// TIA Portal V20 export
// export: Created 2025-12-01T14:57:31.8385946Z, ExportSetting None, DisplayName Totally Integrated Automation Portal, DisplayVersion V20 Update 3, DisplayName TIA Portal Openness, DisplayVersion V20 Update 3, DisplayName TIA Portal Version Control Interface, DisplayVersion V20 Update 3, DisplayName STEP 7 Professional, DisplayVersion V20 Update 3, DisplayName STEP 7 Safety, DisplayVersion V20 Update 2, DisplayName WinCC Basic/Comfort/Advanced, DisplayVersion V20 Update 3, DisplayName WinCC Professional, DisplayVersion V20 Update 3, DisplayName WinCC Unified, DisplayVersion V20 Update 3
FUNCTION_BLOCK "FB531_Ordenes_ELEV / VTD"   // FB531, LAD
{ S7_Optimized_Access := 'FALSE' }
// stored: AutoNumber false, SetENOAutomatically false
   VAR_INPUT
      Estado_CBx : "EstadoZona";   // Estado de la Zona
      Maquina { ExternalVisible := 'False'; ExternalWritable := 'False'} : UInt;   // Numero de Máquina
      Error_Tx : Bool;
   END_VAR
   VAR_OUTPUT
      PosicionDestino : Real;
      Orden : Bool;
   END_VAR
   VAR
      PeticionPiso_Activa { ExternalAccessible := 'False'; ExternalVisible := 'False'; ExternalWritable := 'False'} : Bool;
      Mesa_AVTF_Activo : UInt;
      Mesa_DeDescarga : UInt;
      Mesa { ExternalAccessible := 'False'; ExternalVisible := 'False'; ExternalWritable := 'False'} : UInt;
      Mesa_H1 { ExternalAccessible := 'False'; ExternalVisible := 'False'; ExternalWritable := 'False'} : Bool;   // Orden de Descarga Horquilla/Mesa 1
      Mesa_H2 { ExternalAccessible := 'False'; ExternalVisible := 'False'; ExternalWritable := 'False'} : Bool;   // Orden de Descarga Horquilla/Mesa 2
      AVTF_Activo { ExternalAccessible := 'False'; ExternalVisible := 'False'; ExternalWritable := 'False'} : Bool;   // Orden de Carga hacia la Máquina
      OperacionJdT : Bool;
      Posicion_Destino { ExternalAccessible := 'False'; ExternalVisible := 'False'; ExternalWritable := 'False'} : Real;
      MesaDestino : UInt;
      Rem_MesaDestino : UInt;
      Rem_MesaOrigen : UInt;
   END_VAR
   VAR_TEMP
      OrdenJdT : Struct
         Operacion : UInt;
         MesaHorquilla : UInt;
         MesaCargaDesCarga : UInt;
         VarMesaHorquilla : UInt;
         VarMesaCargaDesCarga : UInt;
      END_STRUCT;
      PrimeraUT_EnMesa : UInt;
      NumMaquina : UInt;
      Mesa_1 : UInt;   // Horquilla/Mesa 1 de la máquina
      Mesa_2 : UInt;   // Horquilla/Mesa 2 de la máquina
      Cero : Byte;
      ValorReturn : Int;
   END_VAR
   VAR_TEMP   // added for the SCL form of the ladder/FBD networks
      _w1 : Bool;
      _w2 : Bool;
      _w3 : Bool;
   END_VAR
BEGIN

REGION Network 1 (SCL): INICIALIZACION
   #Posicion_Destino := 0;

   // Incializar temporales
   #PrimeraUT_EnMesa := 0;

   // Configugracion 
   #Mesa_1 := #NumMaquina :="DB885_ConfigMaquinas".Maquina[#Maquina].Mesa_1;
   #Mesa_2 := "DB885_ConfigMaquinas".Maquina[#Maquina].Mesa_2;

   /// Recoger ordens de JdT
   #OrdenJdT.Operacion := "DB832_Maquinas".Maquinas[#NumMaquina].VTD_ELEV.Operacion;
   #OrdenJdT.MesaHorquilla := "DB832_Maquinas".Maquinas[#NumMaquina].VTD_ELEV.MesaHorquilla ;
   #OrdenJdT.MesaCargaDesCarga := "DB832_Maquinas".Maquinas[#NumMaquina].VTD_ELEV.MesaCargaDesCarga;
   #OrdenJdT.VarMesaHorquilla := #OrdenJdT.MesaHorquilla - "CTE_OffsetMesa";
   #OrdenJdT.VarMesaCargaDesCarga := #OrdenJdT.MesaCargaDesCarga - "CTE_OffsetMesa";
END_REGION

REGION Network 2: >>>>>>>>>>>>>>>>>>>>>>>>>>>>>>>>>>>>>>>>>>>>>>>>>>>>>>>>>>>>>>>>>>>>>>>>>>>>>>>>
END_REGION

REGION Network 3 (SCL): CARGA DEL VTD
   //Si la zona no esta en Marcha o alguna mesa de la maquina esta en error -> No se hace nada 
   IF #Estado_CBx.Marcha_CBx AND #Error_Tx = FALSE THEN
       FOR #Mesa := 1 TO 500 BY 1 DO

           //Si se esta ejecutando una orden anterior no hacemos nada
           IF ((#OperacionJdT = FALSE) AND (#AVTF_Activo = FALSE) AND (#Mesa_H1 = FALSE) AND (#Mesa_H2 = FALSE)) THEN

               // Repasamos todas las mesas de acometida por si alguna tiene activo el AVTF     
               IF (("DB951_InterlockMaquinas".Maquina[#Maquina].Mesa[#Mesa].Out.AVTF) AND ("DB951_InterlockMaquinas".Maquina[#Maquina].Mesa[#Mesa].PosOK_H1 = FALSE) AND ("DB951_InterlockMaquinas".Maquina[#Maquina].Mesa[#Mesa].PosOK_H2 = FALSE)) THEN
                   #PrimeraUT_EnMesa := "DB810_ColasMesas".Colas[#Mesa_AVTF_Activo].UT_PrimeraMesa;
                   #MesaDestino := "DB812_UTs_Control".UT[#PrimeraUT_EnMesa].MesaDestino - "CTE_OffsetMesa";

                   // Revisamos si la mesa destino esta vacia
                   IF "DB900_Estado_Mesas".EstadoVI[#MesaDestino].Etapa_Vacia THEN
                       #Mesa_AVTF_Activo := #Mesa; // Guardamos la mesa que tiene el Aviso Activo
                       #AVTF_Activo := TRUE; 
                       EXIT;
                   END_IF;

               END_IF;
           END_IF;
       END_FOR;
   END_IF;
END_REGION

REGION Network 4: RESETEO SEÑALES CARGA DEL VTD
   // Si en una de las horquillas hay un error y la mesa de Destino se carga mientras resolvemos el error hay que resetear también.
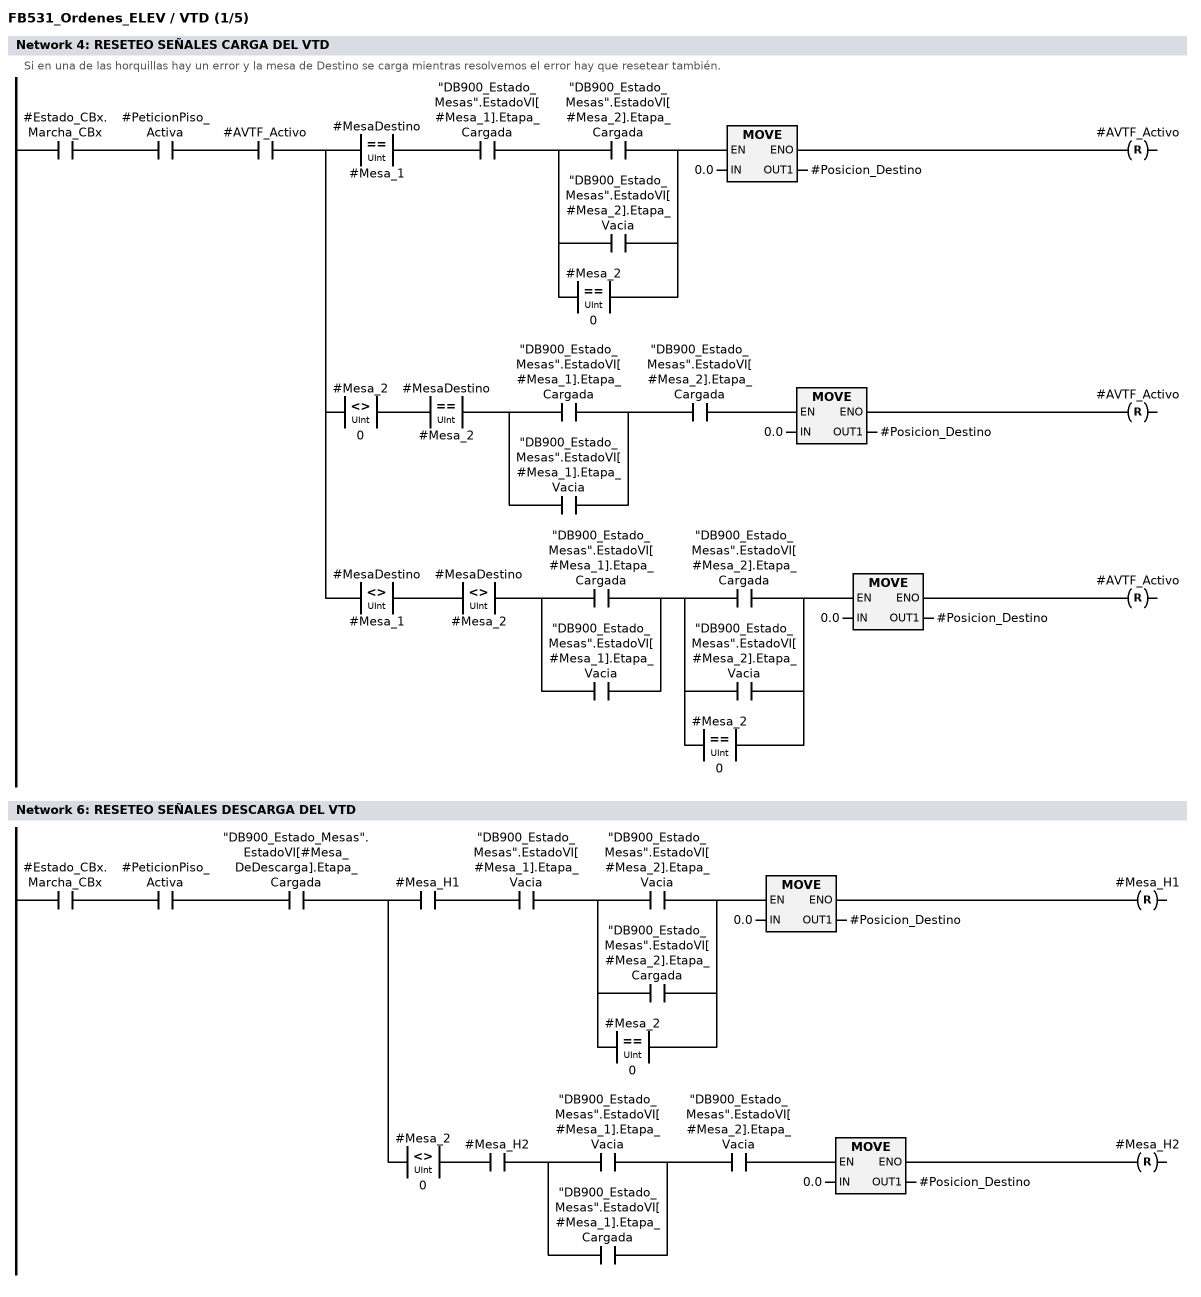
   RUNG wire#powerrail
      Contact( #Estado_CBx.Marcha_CBx )
      Contact( #PeticionPiso_Activa )
      Contact( #AVTF_Activo )
      wire#w1
      { S7_Templates := "SrcType := UInt" } EQ_Contact(in1 := #MesaDestino, in2 := #Mesa_1)
      Contact( "DB900_Estado_Mesas".EstadoVI[#Mesa_1].Etapa_Cargada )
      wire#w2
      Contact( "DB900_Estado_Mesas".EstadoVI[#Mesa_2].Etapa_Cargada )
      wire#w3
      Move(in := 0.0, out1 => #Posicion_Destino)
      R_Coil( #AVTF_Activo )
   END_RUNG
   RUNG wire#w2
      Contact( "DB900_Estado_Mesas".EstadoVI[#Mesa_2].Etapa_Vacia )
   END_RUNG wire#w3
   RUNG wire#w2
      { S7_Templates := "SrcType := UInt" } EQ_Contact(in1 := #Mesa_2, in2 := 0)
   END_RUNG wire#w3
   RUNG wire#w1
      { S7_Templates := "SrcType := UInt" } NE_Contact(in1 := #Mesa_2, in2 := 0)
      { S7_Templates := "SrcType := UInt" } EQ_Contact(in1 := #MesaDestino, in2 := #Mesa_2)
      wire#w4
      Contact( "DB900_Estado_Mesas".EstadoVI[#Mesa_1].Etapa_Cargada )
      wire#w5
      Contact( "DB900_Estado_Mesas".EstadoVI[#Mesa_2].Etapa_Cargada )
      Move(in := 0.0, out1 => #Posicion_Destino)
      R_Coil( #AVTF_Activo )
   END_RUNG
   RUNG wire#w4
      Contact( "DB900_Estado_Mesas".EstadoVI[#Mesa_1].Etapa_Vacia )
   END_RUNG wire#w5
   RUNG wire#w1
      { S7_Templates := "SrcType := UInt" } NE_Contact(in1 := #MesaDestino, in2 := #Mesa_1)
      { S7_Templates := "SrcType := UInt" } NE_Contact(in1 := #MesaDestino, in2 := #Mesa_2)
      wire#w6
      Contact( "DB900_Estado_Mesas".EstadoVI[#Mesa_1].Etapa_Cargada )
      wire#w7
      Contact( "DB900_Estado_Mesas".EstadoVI[#Mesa_2].Etapa_Cargada )
      wire#w8
      Move(in := 0.0, out1 => #Posicion_Destino)
      R_Coil( #AVTF_Activo )
   END_RUNG
   RUNG wire#w6
      Contact( "DB900_Estado_Mesas".EstadoVI[#Mesa_1].Etapa_Vacia )
   END_RUNG wire#w7
   RUNG wire#w7
      Contact( "DB900_Estado_Mesas".EstadoVI[#Mesa_2].Etapa_Vacia )
   END_RUNG wire#w8
   RUNG wire#w7
      { S7_Templates := "SrcType := UInt" } EQ_Contact(in1 := #Mesa_2, in2 := 0)
   END_RUNG wire#w8
   // the same network as SCL:
   #_w1 := #Estado_CBx.Marcha_CBx AND #PeticionPiso_Activa AND #AVTF_Activo;
   IF #_w1 AND (#MesaDestino = #Mesa_1) AND "DB900_Estado_Mesas".EstadoVI[#Mesa_1].Etapa_Cargada AND ("DB900_Estado_Mesas".EstadoVI[#Mesa_2].Etapa_Cargada OR "DB900_Estado_Mesas".EstadoVI[#Mesa_2].Etapa_Vacia OR (#Mesa_2 = 0)) THEN
       #Posicion_Destino := 0.0;
       #AVTF_Activo := FALSE;
   END_IF;
   IF #_w1 AND (#Mesa_2 <> 0) AND (#MesaDestino = #Mesa_2) AND ("DB900_Estado_Mesas".EstadoVI[#Mesa_1].Etapa_Cargada OR "DB900_Estado_Mesas".EstadoVI[#Mesa_1].Etapa_Vacia) AND "DB900_Estado_Mesas".EstadoVI[#Mesa_2].Etapa_Cargada THEN
       #Posicion_Destino := 0.0;
       #AVTF_Activo := FALSE;
   END_IF;
   IF #_w1 AND (#MesaDestino <> #Mesa_1) AND (#MesaDestino <> #Mesa_2) AND ("DB900_Estado_Mesas".EstadoVI[#Mesa_1].Etapa_Cargada OR "DB900_Estado_Mesas".EstadoVI[#Mesa_1].Etapa_Vacia) AND ("DB900_Estado_Mesas".EstadoVI[#Mesa_2].Etapa_Cargada OR "DB900_Estado_Mesas".EstadoVI[#Mesa_2].Etapa_Vacia OR (#Mesa_2 = 0)) THEN
       #Posicion_Destino := 0.0;
       #AVTF_Activo := FALSE;
   END_IF;
END_REGION

REGION Network 5 (SCL): DESCARGA DEL VTD
   //Si la zona no esta en Marcha o alguna mesa de la maquina esta en error -> No se hace nada 
   IF #Estado_CBx.Marcha_CBx = TRUE AND #Error_Tx = FALSE THEN

       //Si se esta ejecutando una orden anterior no hacemos nada
       IF ((#OperacionJdT = FALSE) AND (#AVTF_Activo = FALSE) AND (#Mesa_H1 = FALSE) AND (#Mesa_H2 = FALSE)) THEN

           // Repasamos todas las mesas de acometida por si alguna tiene activo el AVTF     
           IF (("DB900_Estado_Mesas".EstadoVI[#Mesa_1].Etapa_Cargada) AND ("DB951_InterlockMaquinas".Maquina[#Maquina].H1.Out.AVTF_Dcha OR "DB951_InterlockMaquinas".Maquina[#Maquina].H1.Out.AVTF_Izq)) THEN
               #PrimeraUT_EnMesa := "DB810_ColasMesas".Colas[#Mesa_1].UT_PrimeraMesa;
               #Mesa_DeDescarga := "DB812_UTs_Control".UT[#PrimeraUT_EnMesa].MesaDestino - "CTE_OffsetMesa";

               // Revisamos si la mesa destino esta vacia
               IF "DB900_Estado_Mesas".EstadoVI[#Mesa_DeDescarga].Etapa_Vacia THEN
                   #Mesa_H1 := TRUE;
               END_IF;

           ELSIF (("DB900_Estado_Mesas".EstadoVI[#Mesa_2].Etapa_Cargada) AND ("DB951_InterlockMaquinas".Maquina[#Maquina].H2.Out.AVTF_Dcha OR "DB951_InterlockMaquinas".Maquina[#Maquina].H2.Out.AVTF_Izq)) THEN
               #PrimeraUT_EnMesa := "DB810_ColasMesas".Colas[#Mesa_2].UT_PrimeraMesa;
               #Mesa_DeDescarga := "DB812_UTs_Control".UT[#PrimeraUT_EnMesa].MesaDestino - "CTE_OffsetMesa";

               // Revisamos si la mesa destino esta vacia
               IF "DB900_Estado_Mesas".EstadoVI[#Mesa_DeDescarga].Etapa_Vacia THEN
                   #Mesa_H2 := TRUE;
               END_IF;

           END_IF;
       END_IF;
   END_IF;
END_REGION

REGION Network 6: RESETEO SEÑALES DESCARGA DEL VTD
   RUNG wire#powerrail
      Contact( #Estado_CBx.Marcha_CBx )
      Contact( #PeticionPiso_Activa )
      Contact( "DB900_Estado_Mesas".EstadoVI[#Mesa_DeDescarga].Etapa_Cargada )
      wire#w1
      Contact( #Mesa_H1 )
      Contact( "DB900_Estado_Mesas".EstadoVI[#Mesa_1].Etapa_Vacia )
      wire#w2
      Contact( "DB900_Estado_Mesas".EstadoVI[#Mesa_2].Etapa_Vacia )
      wire#w3
      Move(in := 0.0, out1 => #Posicion_Destino)
      R_Coil( #Mesa_H1 )
   END_RUNG
   RUNG wire#w2
      Contact( "DB900_Estado_Mesas".EstadoVI[#Mesa_2].Etapa_Cargada )
   END_RUNG wire#w3
   RUNG wire#w2
      { S7_Templates := "SrcType := UInt" } EQ_Contact(in1 := #Mesa_2, in2 := 0)
   END_RUNG wire#w3
   RUNG wire#w1
      { S7_Templates := "SrcType := UInt" } NE_Contact(in1 := #Mesa_2, in2 := 0)
      Contact( #Mesa_H2 )
      wire#w4
      Contact( "DB900_Estado_Mesas".EstadoVI[#Mesa_1].Etapa_Vacia )
      wire#w5
      Contact( "DB900_Estado_Mesas".EstadoVI[#Mesa_2].Etapa_Vacia )
      Move(in := 0.0, out1 => #Posicion_Destino)
      R_Coil( #Mesa_H2 )
   END_RUNG
   RUNG wire#w4
      Contact( "DB900_Estado_Mesas".EstadoVI[#Mesa_1].Etapa_Cargada )
   END_RUNG wire#w5
   // the same network as SCL:
   #_w1 := #Estado_CBx.Marcha_CBx AND #PeticionPiso_Activa AND "DB900_Estado_Mesas".EstadoVI[#Mesa_DeDescarga].Etapa_Cargada;
   IF #_w1 AND #Mesa_H1 AND "DB900_Estado_Mesas".EstadoVI[#Mesa_1].Etapa_Vacia AND ("DB900_Estado_Mesas".EstadoVI[#Mesa_2].Etapa_Vacia OR "DB900_Estado_Mesas".EstadoVI[#Mesa_2].Etapa_Cargada OR (#Mesa_2 = 0)) THEN
       #Posicion_Destino := 0.0;
       #Mesa_H1 := FALSE;
   END_IF;
   IF #_w1 AND (#Mesa_2 <> 0) AND #Mesa_H2 AND ("DB900_Estado_Mesas".EstadoVI[#Mesa_1].Etapa_Vacia OR "DB900_Estado_Mesas".EstadoVI[#Mesa_1].Etapa_Cargada) AND "DB900_Estado_Mesas".EstadoVI[#Mesa_2].Etapa_Vacia THEN
       #Posicion_Destino := 0.0;
       #Mesa_H2 := FALSE;
   END_IF;
END_REGION

REGION Network 7: >>>>>>>>>>>>>>>>>>>>>>>>>>>>>>>>>>>>>>>>>>>>>>>>>>>>>>>>>>>>>>>>>>>>>>>>>>>>>>>>
END_REGION

REGION Network 8: Activamos las peticiones para mover la maquina
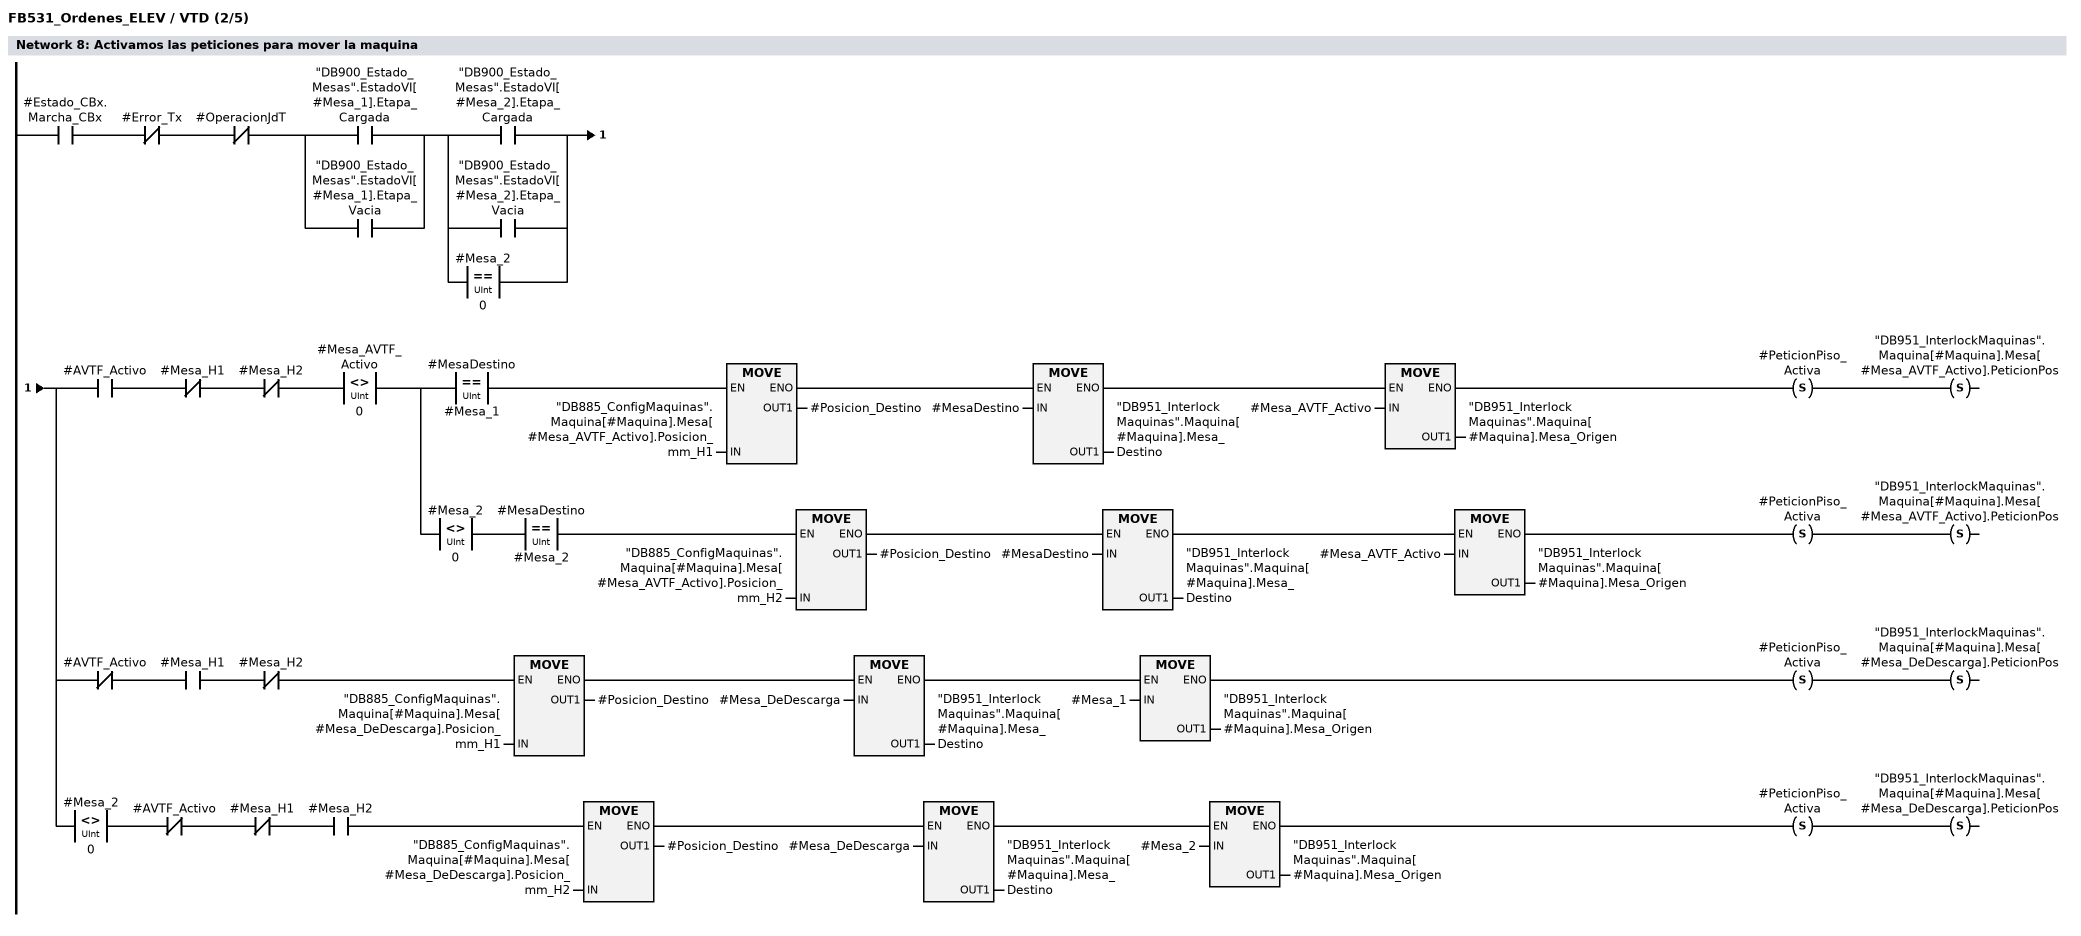
   RUNG wire#powerrail
      Contact( #Estado_CBx.Marcha_CBx )
      I_Contact( #Error_Tx )
      I_Contact( #OperacionJdT )
      wire#w1
      Contact( "DB900_Estado_Mesas".EstadoVI[#Mesa_1].Etapa_Cargada )
      wire#w2
      Contact( "DB900_Estado_Mesas".EstadoVI[#Mesa_2].Etapa_Cargada )
      wire#w3
      Contact( #AVTF_Activo )
      I_Contact( #Mesa_H1 )
      I_Contact( #Mesa_H2 )
      { S7_Templates := "SrcType := UInt" } NE_Contact(in1 := #Mesa_AVTF_Activo, in2 := 0)
      wire#w4
      { S7_Templates := "SrcType := UInt" } EQ_Contact(in1 := #MesaDestino, in2 := #Mesa_1)
      Move(in := "DB885_ConfigMaquinas".Maquina[#Maquina].Mesa[#Mesa_AVTF_Activo].Posicion_mm_H1, out1 => #Posicion_Destino)
      Move(in := #MesaDestino, out1 => "DB951_InterlockMaquinas".Maquina[#Maquina].Mesa_Destino)
      Move(in := #Mesa_AVTF_Activo, out1 => "DB951_InterlockMaquinas".Maquina[#Maquina].Mesa_Origen)
      S_Coil( #PeticionPiso_Activa )
      S_Coil( "DB951_InterlockMaquinas".Maquina[#Maquina].Mesa[#Mesa_AVTF_Activo].PeticionPos )
   END_RUNG
   RUNG wire#w1
      Contact( "DB900_Estado_Mesas".EstadoVI[#Mesa_1].Etapa_Vacia )
   END_RUNG wire#w2
   RUNG wire#w2
      Contact( "DB900_Estado_Mesas".EstadoVI[#Mesa_2].Etapa_Vacia )
   END_RUNG wire#w3
   RUNG wire#w2
      { S7_Templates := "SrcType := UInt" } EQ_Contact(in1 := #Mesa_2, in2 := 0)
   END_RUNG wire#w3
   RUNG wire#w4
      { S7_Templates := "SrcType := UInt" } NE_Contact(in1 := #Mesa_2, in2 := 0)
      { S7_Templates := "SrcType := UInt" } EQ_Contact(in1 := #MesaDestino, in2 := #Mesa_2)
      Move(in := "DB885_ConfigMaquinas".Maquina[#Maquina].Mesa[#Mesa_AVTF_Activo].Posicion_mm_H2, out1 => #Posicion_Destino)
      Move(in := #MesaDestino, out1 => "DB951_InterlockMaquinas".Maquina[#Maquina].Mesa_Destino)
      Move(in := #Mesa_AVTF_Activo, out1 => "DB951_InterlockMaquinas".Maquina[#Maquina].Mesa_Origen)
      S_Coil( #PeticionPiso_Activa )
      S_Coil( "DB951_InterlockMaquinas".Maquina[#Maquina].Mesa[#Mesa_AVTF_Activo].PeticionPos )
   END_RUNG
   RUNG wire#w3
      I_Contact( #AVTF_Activo )
      Contact( #Mesa_H1 )
      I_Contact( #Mesa_H2 )
      Move(in := "DB885_ConfigMaquinas".Maquina[#Maquina].Mesa[#Mesa_DeDescarga].Posicion_mm_H1, out1 => #Posicion_Destino)
      Move(in := #Mesa_DeDescarga, out1 => "DB951_InterlockMaquinas".Maquina[#Maquina].Mesa_Destino)
      Move(in := #Mesa_1, out1 => "DB951_InterlockMaquinas".Maquina[#Maquina].Mesa_Origen)
      S_Coil( #PeticionPiso_Activa )
      S_Coil( "DB951_InterlockMaquinas".Maquina[#Maquina].Mesa[#Mesa_DeDescarga].PeticionPos )
   END_RUNG
   RUNG wire#w3
      { S7_Templates := "SrcType := UInt" } NE_Contact(in1 := #Mesa_2, in2 := 0)
      I_Contact( #AVTF_Activo )
      I_Contact( #Mesa_H1 )
      Contact( #Mesa_H2 )
      Move(in := "DB885_ConfigMaquinas".Maquina[#Maquina].Mesa[#Mesa_DeDescarga].Posicion_mm_H2, out1 => #Posicion_Destino)
      Move(in := #Mesa_DeDescarga, out1 => "DB951_InterlockMaquinas".Maquina[#Maquina].Mesa_Destino)
      Move(in := #Mesa_2, out1 => "DB951_InterlockMaquinas".Maquina[#Maquina].Mesa_Origen)
      S_Coil( #PeticionPiso_Activa )
      S_Coil( "DB951_InterlockMaquinas".Maquina[#Maquina].Mesa[#Mesa_DeDescarga].PeticionPos )
   END_RUNG
   // the same network as SCL:
   #_w1 := #Estado_CBx.Marcha_CBx AND NOT #Error_Tx AND NOT #OperacionJdT AND ("DB900_Estado_Mesas".EstadoVI[#Mesa_1].Etapa_Cargada OR "DB900_Estado_Mesas".EstadoVI[#Mesa_1].Etapa_Vacia) AND ("DB900_Estado_Mesas".EstadoVI[#Mesa_2].Etapa_Cargada OR "DB900_Estado_Mesas".EstadoVI[#Mesa_2].Etapa_Vacia OR (#Mesa_2 = 0));
   #_w2 := #_w1 AND #AVTF_Activo AND NOT #Mesa_H1 AND NOT #Mesa_H2 AND (#Mesa_AVTF_Activo <> 0);
   IF #_w2 AND (#MesaDestino = #Mesa_1) THEN
       #Posicion_Destino := "DB885_ConfigMaquinas".Maquina[#Maquina].Mesa[#Mesa_AVTF_Activo].Posicion_mm_H1;
       "DB951_InterlockMaquinas".Maquina[#Maquina].Mesa_Destino := #MesaDestino;
       "DB951_InterlockMaquinas".Maquina[#Maquina].Mesa_Origen := #Mesa_AVTF_Activo;
       #PeticionPiso_Activa := TRUE;
       "DB951_InterlockMaquinas".Maquina[#Maquina].Mesa[#Mesa_AVTF_Activo].PeticionPos := TRUE;
   END_IF;
   IF #_w2 AND (#Mesa_2 <> 0) AND (#MesaDestino = #Mesa_2) THEN
       #Posicion_Destino := "DB885_ConfigMaquinas".Maquina[#Maquina].Mesa[#Mesa_AVTF_Activo].Posicion_mm_H2;
       "DB951_InterlockMaquinas".Maquina[#Maquina].Mesa_Destino := #MesaDestino;
       "DB951_InterlockMaquinas".Maquina[#Maquina].Mesa_Origen := #Mesa_AVTF_Activo;
       #PeticionPiso_Activa := TRUE;
       "DB951_InterlockMaquinas".Maquina[#Maquina].Mesa[#Mesa_AVTF_Activo].PeticionPos := TRUE;
   END_IF;
   IF #_w1 AND NOT #AVTF_Activo AND #Mesa_H1 AND NOT #Mesa_H2 THEN
       #Posicion_Destino := "DB885_ConfigMaquinas".Maquina[#Maquina].Mesa[#Mesa_DeDescarga].Posicion_mm_H1;
       "DB951_InterlockMaquinas".Maquina[#Maquina].Mesa_Destino := #Mesa_DeDescarga;
       "DB951_InterlockMaquinas".Maquina[#Maquina].Mesa_Origen := #Mesa_1;
       #PeticionPiso_Activa := TRUE;
       "DB951_InterlockMaquinas".Maquina[#Maquina].Mesa[#Mesa_DeDescarga].PeticionPos := TRUE;
   END_IF;
   IF #_w1 AND (#Mesa_2 <> 0) AND NOT #AVTF_Activo AND NOT #Mesa_H1 AND #Mesa_H2 THEN
       #Posicion_Destino := "DB885_ConfigMaquinas".Maquina[#Maquina].Mesa[#Mesa_DeDescarga].Posicion_mm_H2;
       "DB951_InterlockMaquinas".Maquina[#Maquina].Mesa_Destino := #Mesa_DeDescarga;
       "DB951_InterlockMaquinas".Maquina[#Maquina].Mesa_Origen := #Mesa_2;
       #PeticionPiso_Activa := TRUE;
       "DB951_InterlockMaquinas".Maquina[#Maquina].Mesa[#Mesa_DeDescarga].PeticionPos := TRUE;
   END_IF;
END_REGION

REGION Network 9: >>>>>>>>>>>>>>>>>>>>>>>>>>>>>>>>>>>>>>>>>>>>>>>>>>>>>>>>>>>>>>>>>>>>>>>>>>>>>>>>
END_REGION

REGION Network 10: SET >>> Operaciones desde JDT
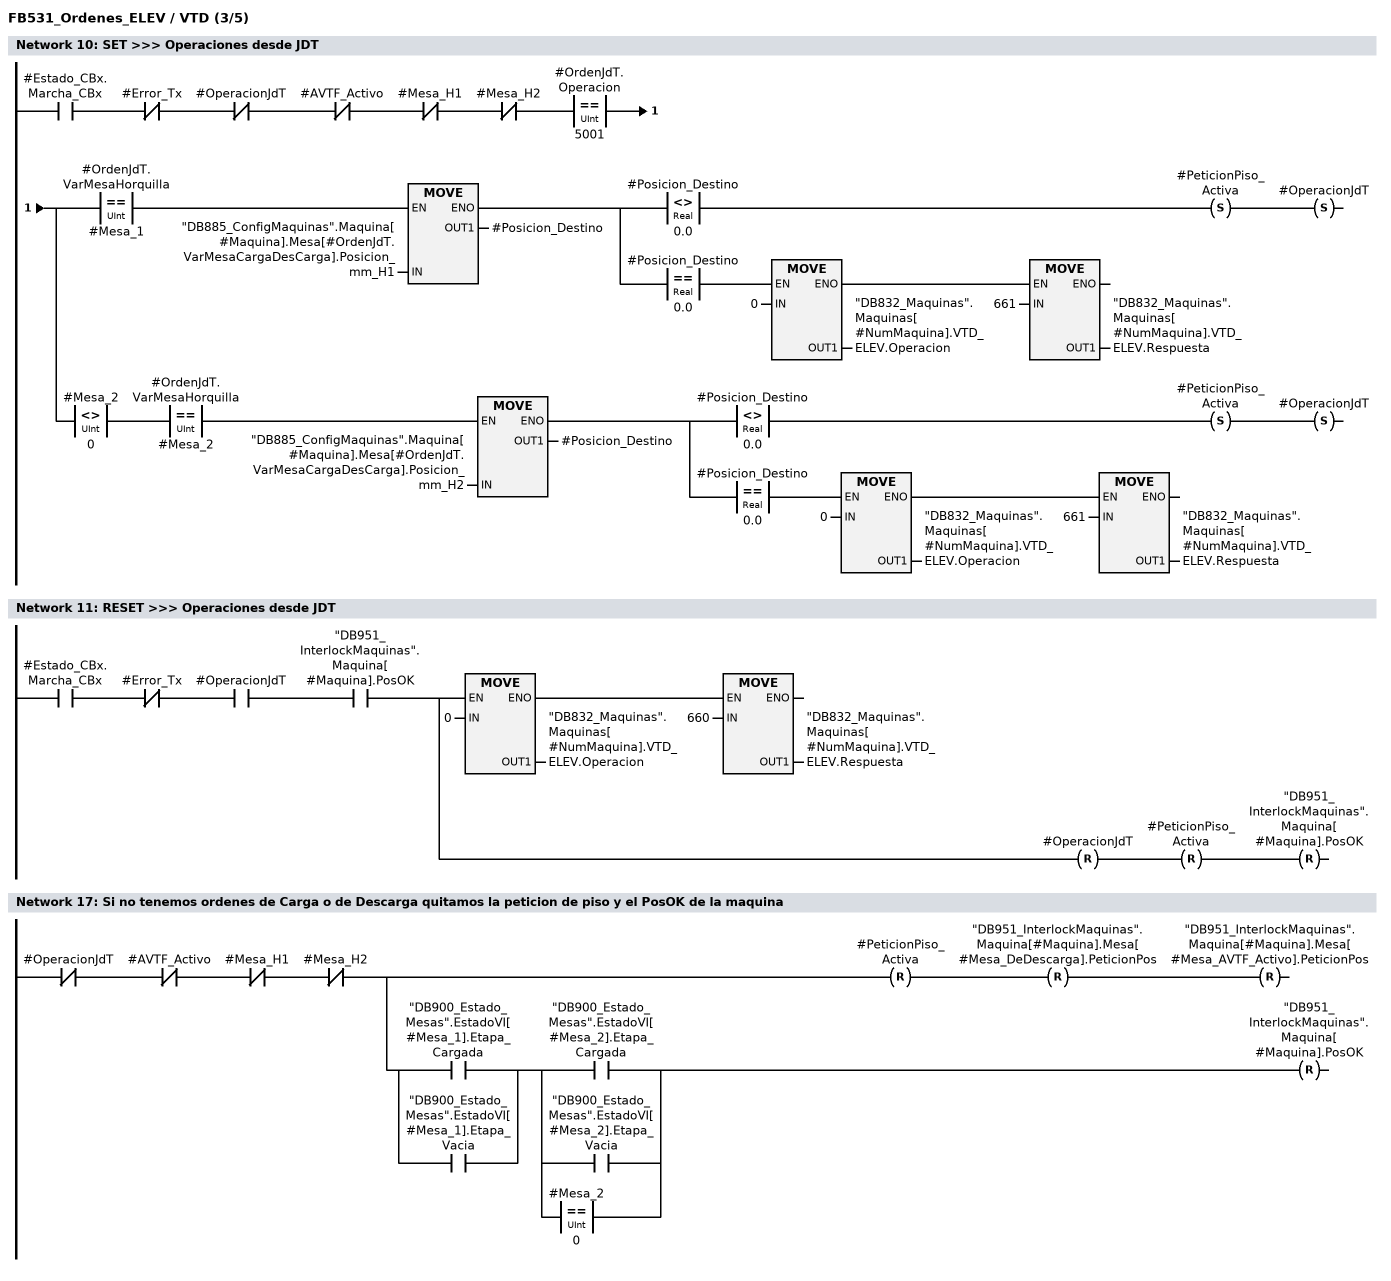
   RUNG wire#powerrail
      Contact( #Estado_CBx.Marcha_CBx )
      I_Contact( #Error_Tx )
      I_Contact( #OperacionJdT )
      I_Contact( #AVTF_Activo )
      I_Contact( #Mesa_H1 )
      I_Contact( #Mesa_H2 )
      { S7_Templates := "SrcType := UInt" } EQ_Contact(in1 := #OrdenJdT.Operacion, in2 := 5001)
      wire#w1
      { S7_Templates := "SrcType := UInt" } EQ_Contact(in1 := #OrdenJdT.VarMesaHorquilla, in2 := #Mesa_1)
      Move(in := "DB885_ConfigMaquinas".Maquina[#Maquina].Mesa[#OrdenJdT.VarMesaCargaDesCarga].Posicion_mm_H1, out1 => #Posicion_Destino)
      wire#w2
      { S7_Templates := "SrcType := Real" } NE_Contact(in1 := #Posicion_Destino, in2 := 0.0)
      S_Coil( #PeticionPiso_Activa )
      S_Coil( #OperacionJdT )
   END_RUNG
   RUNG wire#w2
      { S7_Templates := "SrcType := Real" } EQ_Contact(in1 := #Posicion_Destino, in2 := 0.0)
      Move(in := 0, out1 => "DB832_Maquinas".Maquinas[#NumMaquina].VTD_ELEV.Operacion)
      Move(in := 661, out1 => "DB832_Maquinas".Maquinas[#NumMaquina].VTD_ELEV.Respuesta)
   END_RUNG
   RUNG wire#w1
      { S7_Templates := "SrcType := UInt" } NE_Contact(in1 := #Mesa_2, in2 := 0)
      { S7_Templates := "SrcType := UInt" } EQ_Contact(in1 := #OrdenJdT.VarMesaHorquilla, in2 := #Mesa_2)
      Move(in := "DB885_ConfigMaquinas".Maquina[#Maquina].Mesa[#OrdenJdT.VarMesaCargaDesCarga].Posicion_mm_H2, out1 => #Posicion_Destino)
      wire#w3
      { S7_Templates := "SrcType := Real" } NE_Contact(in1 := #Posicion_Destino, in2 := 0.0)
      S_Coil( #PeticionPiso_Activa )
      S_Coil( #OperacionJdT )
   END_RUNG
   RUNG wire#w3
      { S7_Templates := "SrcType := Real" } EQ_Contact(in1 := #Posicion_Destino, in2 := 0.0)
      Move(in := 0, out1 => "DB832_Maquinas".Maquinas[#NumMaquina].VTD_ELEV.Operacion)
      Move(in := 661, out1 => "DB832_Maquinas".Maquinas[#NumMaquina].VTD_ELEV.Respuesta)
   END_RUNG
   // the same network as SCL:
   #_w1 := #Estado_CBx.Marcha_CBx AND NOT #Error_Tx AND NOT #OperacionJdT AND NOT #AVTF_Activo AND NOT #Mesa_H1 AND NOT #Mesa_H2 AND (#OrdenJdT.Operacion = 5001);
   #_w2 := #_w1 AND (#OrdenJdT.VarMesaHorquilla = #Mesa_1);
   IF #_w2 THEN
       #Posicion_Destino := "DB885_ConfigMaquinas".Maquina[#Maquina].Mesa[#OrdenJdT.VarMesaCargaDesCarga].Posicion_mm_H1;
   END_IF;
   IF #_w2 AND (#Posicion_Destino <> 0.0) THEN
       #PeticionPiso_Activa := TRUE;
       #OperacionJdT := TRUE;
   END_IF;
   IF #_w2 AND (#Posicion_Destino = 0.0) THEN
       "DB832_Maquinas".Maquinas[#NumMaquina].VTD_ELEV.Operacion := 0;
       "DB832_Maquinas".Maquinas[#NumMaquina].VTD_ELEV.Respuesta := 661;
   END_IF;
   #_w3 := #_w1 AND (#Mesa_2 <> 0) AND (#OrdenJdT.VarMesaHorquilla = #Mesa_2);
   IF #_w3 THEN
       #Posicion_Destino := "DB885_ConfigMaquinas".Maquina[#Maquina].Mesa[#OrdenJdT.VarMesaCargaDesCarga].Posicion_mm_H2;
   END_IF;
   IF #_w3 AND (#Posicion_Destino <> 0.0) THEN
       #PeticionPiso_Activa := TRUE;
       #OperacionJdT := TRUE;
   END_IF;
   IF #_w3 AND (#Posicion_Destino = 0.0) THEN
       "DB832_Maquinas".Maquinas[#NumMaquina].VTD_ELEV.Operacion := 0;
       "DB832_Maquinas".Maquinas[#NumMaquina].VTD_ELEV.Respuesta := 661;
   END_IF;
END_REGION

REGION Network 11: RESET >>> Operaciones desde JDT
   RUNG wire#powerrail
      Contact( #Estado_CBx.Marcha_CBx )
      I_Contact( #Error_Tx )
      Contact( #OperacionJdT )
      Contact( "DB951_InterlockMaquinas".Maquina[#Maquina].PosOK )
      wire#w1
      Move(in := 0, out1 => "DB832_Maquinas".Maquinas[#NumMaquina].VTD_ELEV.Operacion)
      Move(in := 660, out1 => "DB832_Maquinas".Maquinas[#NumMaquina].VTD_ELEV.Respuesta)
   END_RUNG
   RUNG wire#w1
      R_Coil( #OperacionJdT )
      R_Coil( #PeticionPiso_Activa )
      R_Coil( "DB951_InterlockMaquinas".Maquina[#Maquina].PosOK )
   END_RUNG
   // the same network as SCL:
   IF #Estado_CBx.Marcha_CBx AND NOT #Error_Tx AND #OperacionJdT AND "DB951_InterlockMaquinas".Maquina[#Maquina].PosOK THEN
       "DB832_Maquinas".Maquinas[#NumMaquina].VTD_ELEV.Operacion := 0;
       "DB832_Maquinas".Maquinas[#NumMaquina].VTD_ELEV.Respuesta := 660;
   END_IF;
   #_w1 := #Estado_CBx.Marcha_CBx AND NOT #Error_Tx AND #OperacionJdT AND "DB951_InterlockMaquinas".Maquina[#Maquina].PosOK;
   IF #_w1 THEN
       #OperacionJdT := FALSE;
       #PeticionPiso_Activa := FALSE;
       "DB951_InterlockMaquinas".Maquina[#Maquina].PosOK := FALSE;
   END_IF;
END_REGION

REGION Network 12: >>>>>>>>>>>>>>>>>>>>>>>>>>>>>>>>>>>>>>>>>>>>>>>>>>>>>>>>>>>>>>>>>>>>>>>>>>>>>>>>
END_REGION

REGION Network 13 (SCL): Inicializar interlock de la maquina

   #Cero := 0;

   #ValorReturn := FILL(BVAL := #Cero, BLK => "DB951_InterlockMaquinas".Maquina[#Maquina].H1.In);
   #ValorReturn := FILL(BVAL := #Cero, BLK => "DB951_InterlockMaquinas".Maquina[#Maquina].H2.In);

   "DB951_InterlockMaquinas".Maquina[#Maquina].H1.Mesa_EntradaDerecha := 0;
   "DB951_InterlockMaquinas".Maquina[#Maquina].H1.Mesa_EntradaIzquierda := 0;
   "DB951_InterlockMaquinas".Maquina[#Maquina].H2.Mesa_EntradaDerecha := 0;
   "DB951_InterlockMaquinas".Maquina[#Maquina].H2.Mesa_EntradaIzquierda := 0;
END_REGION

REGION Network 14 (SCL): Señales para cargar las mesas de la maquina
   FOR #Mesa := 1 TO 500 BY 1 DO

       #ValorReturn := FILL(BVAL := #Cero, BLK => "DB951_InterlockMaquinas".Maquina[#Maquina].Mesa[#Mesa].In);

         IF "DB951_InterlockMaquinas".Maquina[#Maquina].PosOK THEN
               // Repasamos que mesas tienen la misma cota para la Horquilla 1
               IF "DB885_ConfigMaquinas".Maquina[#Maquina].Mesa[#Mesa].Posicion_mm_H1 = #Posicion_Destino AND "DB951_InterlockMaquinas".Maquina[#Maquina].Mesa[#Mesa].PosOK_H1 THEN

                   // Señales de las Mesas posicionadas a la Derecha
                   IF "DB885_ConfigMaquinas".Maquina[#Maquina].Mesa[#Mesa].Derecha THEN
                       // Señales para cargar las mesas de la maquina
                       "DB951_InterlockMaquinas".Maquina[#Maquina].H1.In.AVTF_Dcha := "DB951_InterlockMaquinas".Maquina[#Maquina].Mesa[#Mesa].Out.AVTF;
                       "DB951_InterlockMaquinas".Maquina[#Maquina].H1.In.P_Mens_Dcha := "DB951_InterlockMaquinas".Maquina[#Maquina].Mesa[#Mesa].Out.P_Mens;
                       "DB951_InterlockMaquinas".Maquina[#Maquina].H1.In.DesCargaAct_Dcha := "DB900_Estado_Mesas".EstadoVI[#Mesa].Descarga_Act;

                       "DB951_InterlockMaquinas".Maquina[#Maquina].Mesa[#Mesa].In.PTF := "DB951_InterlockMaquinas".Maquina[#Maquina].H1.Out.PTF_Dcha;
                       "DB951_InterlockMaquinas".Maquina[#Maquina].Mesa[#Mesa].In.FTF := "DB951_InterlockMaquinas".Maquina[#Maquina].H1.Out.FTF_Dcha;
                       "DB951_InterlockMaquinas".Maquina[#Maquina].Mesa[#Mesa].In.CargaAct := "DB900_Estado_Mesas".EstadoVI[#Mesa_1].Etapas_Carga_E1;

                       "DB951_InterlockMaquinas".Maquina[#Maquina].H1.Mesa_EntradaDerecha := #Mesa;

                       // Señales para descargar las mesas de la maquina
                       "DB951_InterlockMaquinas".Maquina[#Maquina].Mesa[#Mesa].In.AVTF := "DB951_InterlockMaquinas".Maquina[#Maquina].H1.Out.AVTF_Dcha;
                       "DB951_InterlockMaquinas".Maquina[#Maquina].Mesa[#Mesa].In.P_Mens := "DB951_InterlockMaquinas".Maquina[#Maquina].H1.Out.P_Mens_Dcha;
                       "DB951_InterlockMaquinas".Maquina[#Maquina].Mesa[#Mesa].In.DesCargaAct := "DB900_Estado_Mesas".EstadoVI[#Mesa_1].Descarga_Act;

                       "DB951_InterlockMaquinas".Maquina[#Maquina].H1.In.PTF_Dcha := "DB951_InterlockMaquinas".Maquina[#Maquina].Mesa[#Mesa].Out.PTF;
                       "DB951_InterlockMaquinas".Maquina[#Maquina].H1.In.FTF_Dcha := "DB951_InterlockMaquinas".Maquina[#Maquina].Mesa[#Mesa].Out.FTF;
                       "DB951_InterlockMaquinas".Maquina[#Maquina].H1.In.CargaAct_Dcha := "DB900_Estado_Mesas".EstadoVI[#Mesa].Etapas_Carga_E1 OR
                                                                                               "DB900_Estado_Mesas".EstadoVI[#Mesa].Etapas_Carga_E2 OR
                                                                                               "DB900_Estado_Mesas".EstadoVI[#Mesa].Etapas_Carga_E3 OR
                                                                                               "DB900_Estado_Mesas".EstadoVI[#Mesa].Etapas_Carga_E4;

                       "DB951_InterlockMaquinas".Maquina[#Maquina].Mesa[#Mesa].MesaEntrada := #Mesa_1;

                   END_IF;

                   // Señales de las Mesas posicionadas a la Izquierda
                   IF "DB885_ConfigMaquinas".Maquina[#Maquina].Mesa[#Mesa].Izquierda THEN
                       // Señales para cargar las mesas de la maquina
                       "DB951_InterlockMaquinas".Maquina[#Maquina].H1.In.AVTF_Izq := "DB951_InterlockMaquinas".Maquina[#Maquina].Mesa[#Mesa].Out.AVTF;
                       "DB951_InterlockMaquinas".Maquina[#Maquina].H1.In.P_Mens_Izq := "DB951_InterlockMaquinas".Maquina[#Maquina].Mesa[#Mesa].Out.P_Mens;
                       "DB951_InterlockMaquinas".Maquina[#Maquina].H1.In.DesCargaAct_Izq := "DB900_Estado_Mesas".EstadoVI[#Mesa].Descarga_Act;

                       "DB951_InterlockMaquinas".Maquina[#Maquina].Mesa[#Mesa].In.PTF := "DB951_InterlockMaquinas".Maquina[#Maquina].H1.Out.PTF_Izq;
                       "DB951_InterlockMaquinas".Maquina[#Maquina].Mesa[#Mesa].In.FTF := "DB951_InterlockMaquinas".Maquina[#Maquina].H1.Out.FTF_Izq;
                       "DB951_InterlockMaquinas".Maquina[#Maquina].Mesa[#Mesa].In.CargaAct := "DB900_Estado_Mesas".EstadoVI[#Mesa_1].Etapas_Carga_E3;

                       "DB951_InterlockMaquinas".Maquina[#Maquina].H1.Mesa_EntradaIzquierda := #Mesa;

                       // Señales para descargar las mesas de la maquina
                       "DB951_InterlockMaquinas".Maquina[#Maquina].Mesa[#Mesa].In.AVTF := "DB951_InterlockMaquinas".Maquina[#Maquina].H1.Out.AVTF_Izq;
                       "DB951_InterlockMaquinas".Maquina[#Maquina].Mesa[#Mesa].In.P_Mens := "DB951_InterlockMaquinas".Maquina[#Maquina].H1.Out.P_Mens_Izq;
                       "DB951_InterlockMaquinas".Maquina[#Maquina].Mesa[#Mesa].In.DesCargaAct := "DB900_Estado_Mesas".EstadoVI[#Mesa_1].Descarga_Act;

                       "DB951_InterlockMaquinas".Maquina[#Maquina].H1.In.PTF_Izq := "DB951_InterlockMaquinas".Maquina[#Maquina].Mesa[#Mesa].Out.PTF;
                       "DB951_InterlockMaquinas".Maquina[#Maquina].H1.In.FTF_Izq := "DB951_InterlockMaquinas".Maquina[#Maquina].Mesa[#Mesa].Out.FTF;
                       "DB951_InterlockMaquinas".Maquina[#Maquina].H1.In.CargaAct_Izq := "DB900_Estado_Mesas".EstadoVI[#Mesa].Etapas_Carga_E1 OR
                                                                                               "DB900_Estado_Mesas".EstadoVI[#Mesa].Etapas_Carga_E2 OR
                                                                                               "DB900_Estado_Mesas".EstadoVI[#Mesa].Etapas_Carga_E3 OR
                                                                                               "DB900_Estado_Mesas".EstadoVI[#Mesa].Etapas_Carga_E4;

                       "DB951_InterlockMaquinas".Maquina[#Maquina].Mesa[#Mesa].MesaEntrada := #Mesa_1;
                   END_IF;

               END_IF;

               // Repasamos que mesas tienen la misma cota para la Horquilla 2
               IF "DB885_ConfigMaquinas".Maquina[#Maquina].Mesa[#Mesa].Posicion_mm_H2 = #Posicion_Destino AND "DB951_InterlockMaquinas".Maquina[#Maquina].Mesa[#Mesa].PosOK_H2 THEN

                   // Señales de las Mesas posicionadas a la Derecha
                   IF "DB885_ConfigMaquinas".Maquina[#Maquina].Mesa[#Mesa].Derecha THEN
                       // Señales para cargar las mesas de la maquina
                       "DB951_InterlockMaquinas".Maquina[#Maquina].H2.In.AVTF_Dcha := "DB951_InterlockMaquinas".Maquina[#Maquina].Mesa[#Mesa].Out.AVTF;
                       "DB951_InterlockMaquinas".Maquina[#Maquina].H2.In.P_Mens_Dcha := "DB951_InterlockMaquinas".Maquina[#Maquina].Mesa[#Mesa].Out.P_Mens;
                       "DB951_InterlockMaquinas".Maquina[#Maquina].H2.In.DesCargaAct_Dcha := "DB900_Estado_Mesas".EstadoVI[#Mesa].Descarga_Act;

                       "DB951_InterlockMaquinas".Maquina[#Maquina].Mesa[#Mesa].In.PTF := "DB951_InterlockMaquinas".Maquina[#Maquina].H2.Out.PTF_Dcha;
                       "DB951_InterlockMaquinas".Maquina[#Maquina].Mesa[#Mesa].In.FTF := "DB951_InterlockMaquinas".Maquina[#Maquina].H2.Out.FTF_Dcha;
                       "DB951_InterlockMaquinas".Maquina[#Maquina].Mesa[#Mesa].In.CargaAct := "DB900_Estado_Mesas".EstadoVI[#Mesa_2].Etapas_Carga_E1;

                       "DB951_InterlockMaquinas".Maquina[#Maquina].H2.Mesa_EntradaDerecha := #Mesa;

                       // Señales para descargar las mesas de la maquina
                       "DB951_InterlockMaquinas".Maquina[#Maquina].Mesa[#Mesa].In.AVTF := "DB951_InterlockMaquinas".Maquina[#Maquina].H2.Out.AVTF_Dcha;
                       "DB951_InterlockMaquinas".Maquina[#Maquina].Mesa[#Mesa].In.P_Mens := "DB951_InterlockMaquinas".Maquina[#Maquina].H2.Out.P_Mens_Dcha;
                       "DB951_InterlockMaquinas".Maquina[#Maquina].Mesa[#Mesa].In.DesCargaAct := "DB900_Estado_Mesas".EstadoVI[#Mesa_2].Descarga_Act;

                       "DB951_InterlockMaquinas".Maquina[#Maquina].H2.In.PTF_Dcha := "DB951_InterlockMaquinas".Maquina[#Maquina].Mesa[#Mesa].Out.PTF;
                       "DB951_InterlockMaquinas".Maquina[#Maquina].H2.In.FTF_Dcha := "DB951_InterlockMaquinas".Maquina[#Maquina].Mesa[#Mesa].Out.FTF;
                       "DB951_InterlockMaquinas".Maquina[#Maquina].H2.In.CargaAct_Dcha := "DB900_Estado_Mesas".EstadoVI[#Mesa].Etapas_Carga_E1 OR
                                                                                               "DB900_Estado_Mesas".EstadoVI[#Mesa].Etapas_Carga_E2 OR
                                                                                               "DB900_Estado_Mesas".EstadoVI[#Mesa].Etapas_Carga_E3 OR
                                                                                               "DB900_Estado_Mesas".EstadoVI[#Mesa].Etapas_Carga_E4;


                       "DB951_InterlockMaquinas".Maquina[#Maquina].Mesa[#Mesa].MesaEntrada := #Mesa_2;

                   END_IF;

                   // Señales de las Mesas posicionadas a la Izquierda
                   IF "DB885_ConfigMaquinas".Maquina[#Maquina].Mesa[#Mesa].Izquierda THEN
                       // Señales para cargar las mesas de la maquina
                       "DB951_InterlockMaquinas".Maquina[#Maquina].H2.In.AVTF_Izq := "DB951_InterlockMaquinas".Maquina[#Maquina].Mesa[#Mesa].Out.AVTF;
                       "DB951_InterlockMaquinas".Maquina[#Maquina].H2.In.P_Mens_Izq := "DB951_InterlockMaquinas".Maquina[#Maquina].Mesa[#Mesa].Out.P_Mens;
                       "DB951_InterlockMaquinas".Maquina[#Maquina].H2.In.DesCargaAct_Izq := "DB900_Estado_Mesas".EstadoVI[#Mesa].Descarga_Act;

                       "DB951_InterlockMaquinas".Maquina[#Maquina].Mesa[#Mesa].In.PTF := "DB951_InterlockMaquinas".Maquina[#Maquina].H2.Out.PTF_Izq;
                       "DB951_InterlockMaquinas".Maquina[#Maquina].Mesa[#Mesa].In.FTF := "DB951_InterlockMaquinas".Maquina[#Maquina].H2.Out.FTF_Izq;
                       "DB951_InterlockMaquinas".Maquina[#Maquina].Mesa[#Mesa].In.CargaAct := "DB900_Estado_Mesas".EstadoVI[#Mesa_2].Etapas_Carga_E3;

                       "DB951_InterlockMaquinas".Maquina[#Maquina].H2.Mesa_EntradaIzquierda := #Mesa;

                       // Señales para descargar las mesas de la maquina
                       "DB951_InterlockMaquinas".Maquina[#Maquina].Mesa[#Mesa].In.AVTF := "DB951_InterlockMaquinas".Maquina[#Maquina].H2.Out.AVTF_Izq;
                       "DB951_InterlockMaquinas".Maquina[#Maquina].Mesa[#Mesa].In.P_Mens := "DB951_InterlockMaquinas".Maquina[#Maquina].H2.Out.P_Mens_Izq;
                       "DB951_InterlockMaquinas".Maquina[#Maquina].Mesa[#Mesa].In.DesCargaAct := "DB900_Estado_Mesas".EstadoVI[#Mesa_2].Descarga_Act;

                       "DB951_InterlockMaquinas".Maquina[#Maquina].H2.In.PTF_Izq := "DB951_InterlockMaquinas".Maquina[#Maquina].Mesa[#Mesa].Out.PTF;
                       "DB951_InterlockMaquinas".Maquina[#Maquina].H2.In.FTF_Izq := "DB951_InterlockMaquinas".Maquina[#Maquina].Mesa[#Mesa].Out.FTF;
                       "DB951_InterlockMaquinas".Maquina[#Maquina].H2.In.CargaAct_Izq := "DB900_Estado_Mesas".EstadoVI[#Mesa].Etapas_Carga_E1 OR
                                                                                               "DB900_Estado_Mesas".EstadoVI[#Mesa].Etapas_Carga_E2 OR
                                                                                               "DB900_Estado_Mesas".EstadoVI[#Mesa].Etapas_Carga_E3 OR
                                                                                               "DB900_Estado_Mesas".EstadoVI[#Mesa].Etapas_Carga_E4;


                       "DB951_InterlockMaquinas".Maquina[#Maquina].Mesa[#Mesa].MesaEntrada := #Mesa_2;
                   END_IF;
               END_IF;
           END_IF;
       END_FOR;
END_REGION

REGION Network 15: >>>>>>>>>>>>>>>>>>>>>>>>>>>>>>>>>>>>>>>>>>>>>>>>>>>>>>>>>>>>>>>>>>>>>>>>>>>>>>>>
END_REGION

REGION Network 16 (SCL): Activamos el PosOK de todas las mesas que estan en la cota donde ha parado la maquina
   FOR #Mesa := 1 TO 500 BY 1  DO

           "DB951_InterlockMaquinas".Maquina[#Maquina].Mesa[#Mesa].PosOK_H1 := FALSE;
           "DB951_InterlockMaquinas".Maquina[#Maquina].Mesa[#Mesa].PosOK_H2 := FALSE;

           IF #Estado_CBx.Marcha_CBx THEN

               // Repasamos que mesas tienen la misma cota para la Horquilla 1
               IF (("DB885_ConfigMaquinas".Maquina[#Maquina].Mesa[#Mesa].Posicion_mm_H1 = #Posicion_Destino)) THEN

                   // Activamos el PosOK de la Mesa
                   "DB951_InterlockMaquinas".Maquina[#Maquina].Mesa[#Mesa].PosOK_H1 := "DB951_InterlockMaquinas".Maquina[#Maquina].PosOK;

               END_IF;

               // Repasamos que mesas tienen la misma cota para la Horquilla 2
               IF ("DB885_ConfigMaquinas".Maquina[#Maquina].Mesa[#Mesa].Posicion_mm_H2 = #Posicion_Destino) THEN

                   // Activamos el PosOK de la Mesa
                   "DB951_InterlockMaquinas".Maquina[#Maquina].Mesa[#Mesa].PosOK_H2 := "DB951_InterlockMaquinas".Maquina[#Maquina].PosOK;
               END_IF;
           END_IF;
    END_FOR;
END_REGION

REGION Network 17: Si no tenemos ordenes de Carga o de Descarga quitamos la peticion de piso y el PosOK de la maquina
   RUNG wire#powerrail
      I_Contact( #OperacionJdT )
      I_Contact( #AVTF_Activo )
      I_Contact( #Mesa_H1 )
      I_Contact( #Mesa_H2 )
      wire#w1
      R_Coil( #PeticionPiso_Activa )
      R_Coil( "DB951_InterlockMaquinas".Maquina[#Maquina].Mesa[#Mesa_DeDescarga].PeticionPos )
      R_Coil( "DB951_InterlockMaquinas".Maquina[#Maquina].Mesa[#Mesa_AVTF_Activo].PeticionPos )
   END_RUNG
   RUNG wire#w1
      Contact( "DB900_Estado_Mesas".EstadoVI[#Mesa_1].Etapa_Cargada )
      wire#w2
      Contact( "DB900_Estado_Mesas".EstadoVI[#Mesa_2].Etapa_Cargada )
      wire#w3
      R_Coil( "DB951_InterlockMaquinas".Maquina[#Maquina].PosOK )
   END_RUNG
   RUNG wire#w1
      Contact( "DB900_Estado_Mesas".EstadoVI[#Mesa_1].Etapa_Vacia )
   END_RUNG wire#w2
   RUNG wire#w2
      Contact( "DB900_Estado_Mesas".EstadoVI[#Mesa_2].Etapa_Vacia )
   END_RUNG wire#w3
   RUNG wire#w2
      { S7_Templates := "SrcType := UInt" } EQ_Contact(in1 := #Mesa_2, in2 := 0)
   END_RUNG wire#w3
   // the same network as SCL:
   #_w1 := NOT #OperacionJdT AND NOT #AVTF_Activo AND NOT #Mesa_H1 AND NOT #Mesa_H2;
   IF #_w1 THEN
       #PeticionPiso_Activa := FALSE;
       "DB951_InterlockMaquinas".Maquina[#Maquina].Mesa[#Mesa_DeDescarga].PeticionPos := FALSE;
       "DB951_InterlockMaquinas".Maquina[#Maquina].Mesa[#Mesa_AVTF_Activo].PeticionPos := FALSE;
   END_IF;
   IF #_w1 AND ("DB900_Estado_Mesas".EstadoVI[#Mesa_1].Etapa_Cargada OR "DB900_Estado_Mesas".EstadoVI[#Mesa_1].Etapa_Vacia) AND ("DB900_Estado_Mesas".EstadoVI[#Mesa_2].Etapa_Cargada OR "DB900_Estado_Mesas".EstadoVI[#Mesa_2].Etapa_Vacia OR (#Mesa_2 = 0)) THEN
       "DB951_InterlockMaquinas".Maquina[#Maquina].PosOK := FALSE;
   END_IF;
END_REGION

REGION Network 18: Si no estamos en Marcha, reseteamos
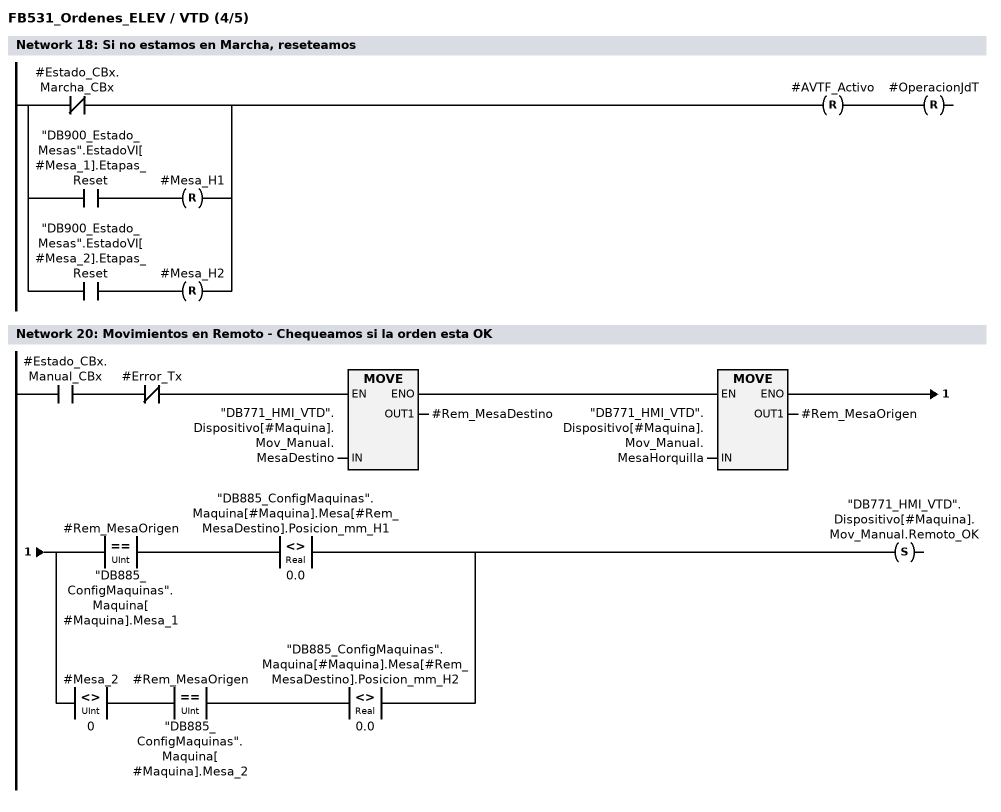
   RUNG wire#powerrail
      I_Contact( #Estado_CBx.Marcha_CBx )
      wire#w1
      R_Coil( #AVTF_Activo )
      R_Coil( #OperacionJdT )
   END_RUNG
   RUNG wire#powerrail
      Contact( "DB900_Estado_Mesas".EstadoVI[#Mesa_1].Etapas_Reset )
      R_Coil( #Mesa_H1 )
   END_RUNG wire#w1
   RUNG wire#powerrail
      Contact( "DB900_Estado_Mesas".EstadoVI[#Mesa_2].Etapas_Reset )
      R_Coil( #Mesa_H2 )
   END_RUNG wire#w1
   // the same network as SCL:
   IF "DB900_Estado_Mesas".EstadoVI[#Mesa_1].Etapas_Reset THEN #Mesa_H1 := FALSE; END_IF;
   IF "DB900_Estado_Mesas".EstadoVI[#Mesa_2].Etapas_Reset THEN #Mesa_H2 := FALSE; END_IF;
   IF NOT #Estado_CBx.Marcha_CBx OR "DB900_Estado_Mesas".EstadoVI[#Mesa_1].Etapas_Reset OR "DB900_Estado_Mesas".EstadoVI[#Mesa_2].Etapas_Reset THEN
       #AVTF_Activo := FALSE;
       #OperacionJdT := FALSE;
   END_IF;
END_REGION

REGION Network 19: >>>>>>>>>>>>>>>>>>>>>>>>>>>>>>>>>>>>>>>>>>>>>>>>>>>>>>>>>>>>>>>>>>>>>>>>>>>>>>>>
END_REGION

REGION Network 20: Movimientos en Remoto - Chequeamos si la orden esta OK
   RUNG wire#powerrail
      Contact( #Estado_CBx.Manual_CBx )
      I_Contact( #Error_Tx )
      Move(in := "DB771_HMI_VTD".Dispositivo[#Maquina].Mov_Manual.MesaDestino, out1 => #Rem_MesaDestino)
      Move(in := "DB771_HMI_VTD".Dispositivo[#Maquina].Mov_Manual.MesaHorquilla, out1 => #Rem_MesaOrigen)
      wire#w1
      { S7_Templates := "SrcType := UInt" } EQ_Contact(in1 := #Rem_MesaOrigen, in2 := "DB885_ConfigMaquinas".Maquina[#Maquina].Mesa_1)
      { S7_Templates := "SrcType := Real" } NE_Contact(in1 := "DB885_ConfigMaquinas".Maquina[#Maquina].Mesa[#Rem_MesaDestino].Posicion_mm_H1, in2 := 0.0)
      wire#w2
      S_Coil( "DB771_HMI_VTD".Dispositivo[#Maquina].Mov_Manual.Remoto_OK )
   END_RUNG
   RUNG wire#w1
      { S7_Templates := "SrcType := UInt" } NE_Contact(in1 := #Mesa_2, in2 := 0)
      { S7_Templates := "SrcType := UInt" } EQ_Contact(in1 := #Rem_MesaOrigen, in2 := "DB885_ConfigMaquinas".Maquina[#Maquina].Mesa_2)
      { S7_Templates := "SrcType := Real" } NE_Contact(in1 := "DB885_ConfigMaquinas".Maquina[#Maquina].Mesa[#Rem_MesaDestino].Posicion_mm_H2, in2 := 0.0)
   END_RUNG wire#w2
   // the same network as SCL:
   #_w1 := #Estado_CBx.Manual_CBx AND NOT #Error_Tx;
   IF #_w1 THEN
       #Rem_MesaDestino := "DB771_HMI_VTD".Dispositivo[#Maquina].Mov_Manual.MesaDestino;
       #Rem_MesaOrigen := "DB771_HMI_VTD".Dispositivo[#Maquina].Mov_Manual.MesaHorquilla;
   END_IF;
   IF #_w1 AND (((#Rem_MesaOrigen = "DB885_ConfigMaquinas".Maquina[#Maquina].Mesa_1) AND ("DB885_ConfigMaquinas".Maquina[#Maquina].Mesa[#Rem_MesaDestino].Posicion_mm_H1 <> 0.0)) OR ((#Mesa_2 <> 0) AND (#Rem_MesaOrigen = "DB885_ConfigMaquinas".Maquina[#Maquina].Mesa_2) AND ("DB885_ConfigMaquinas".Maquina[#Maquina].Mesa[#Rem_MesaDestino].Posicion_mm_H2 <> 0.0))) THEN
       "DB771_HMI_VTD".Dispositivo[#Maquina].Mov_Manual.Remoto_OK := TRUE;
   END_IF;
END_REGION

REGION Network 21: Movimientos en Remoto
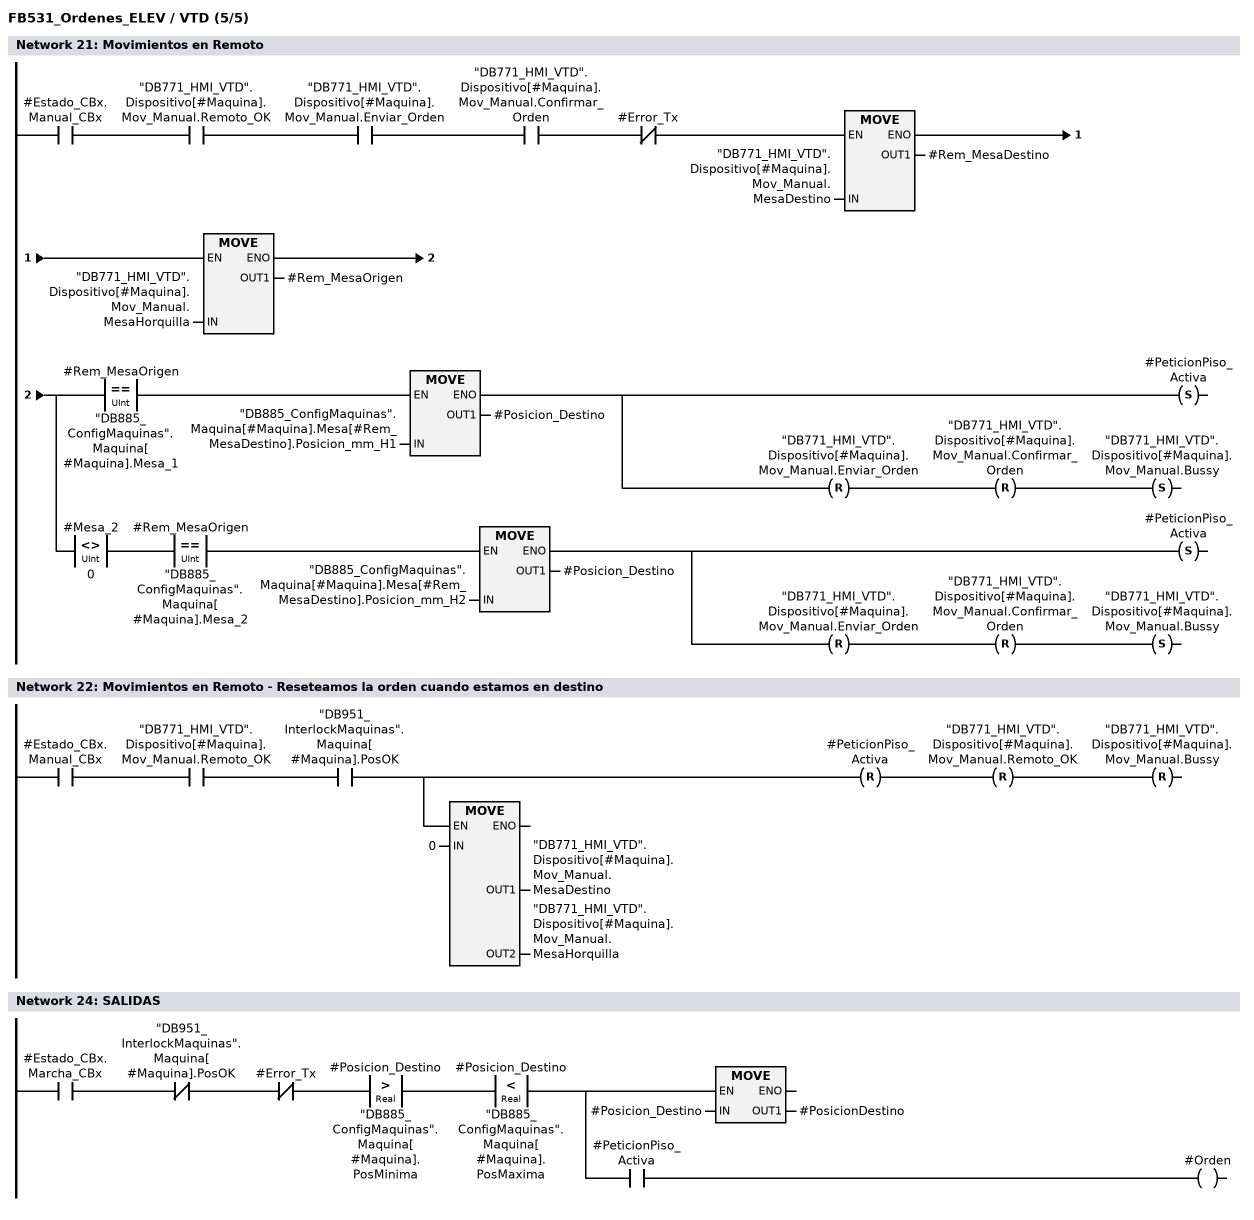
   RUNG wire#powerrail
      Contact( #Estado_CBx.Manual_CBx )
      Contact( "DB771_HMI_VTD".Dispositivo[#Maquina].Mov_Manual.Remoto_OK )
      Contact( "DB771_HMI_VTD".Dispositivo[#Maquina].Mov_Manual.Enviar_Orden )
      Contact( "DB771_HMI_VTD".Dispositivo[#Maquina].Mov_Manual.Confirmar_Orden )
      I_Contact( #Error_Tx )
      Move(in := "DB771_HMI_VTD".Dispositivo[#Maquina].Mov_Manual.MesaDestino, out1 => #Rem_MesaDestino)
      Move(in := "DB771_HMI_VTD".Dispositivo[#Maquina].Mov_Manual.MesaHorquilla, out1 => #Rem_MesaOrigen)
      wire#w1
      { S7_Templates := "SrcType := UInt" } EQ_Contact(in1 := #Rem_MesaOrigen, in2 := "DB885_ConfigMaquinas".Maquina[#Maquina].Mesa_1)
      Move(in := "DB885_ConfigMaquinas".Maquina[#Maquina].Mesa[#Rem_MesaDestino].Posicion_mm_H1, out1 => #Posicion_Destino)
      wire#w2
      S_Coil( #PeticionPiso_Activa )
   END_RUNG
   RUNG wire#w2
      R_Coil( "DB771_HMI_VTD".Dispositivo[#Maquina].Mov_Manual.Enviar_Orden )
      R_Coil( "DB771_HMI_VTD".Dispositivo[#Maquina].Mov_Manual.Confirmar_Orden )
      S_Coil( "DB771_HMI_VTD".Dispositivo[#Maquina].Mov_Manual.Bussy )
   END_RUNG
   RUNG wire#w1
      { S7_Templates := "SrcType := UInt" } NE_Contact(in1 := #Mesa_2, in2 := 0)
      { S7_Templates := "SrcType := UInt" } EQ_Contact(in1 := #Rem_MesaOrigen, in2 := "DB885_ConfigMaquinas".Maquina[#Maquina].Mesa_2)
      Move(in := "DB885_ConfigMaquinas".Maquina[#Maquina].Mesa[#Rem_MesaDestino].Posicion_mm_H2, out1 => #Posicion_Destino)
      wire#w3
      S_Coil( #PeticionPiso_Activa )
   END_RUNG
   RUNG wire#w3
      R_Coil( "DB771_HMI_VTD".Dispositivo[#Maquina].Mov_Manual.Enviar_Orden )
      R_Coil( "DB771_HMI_VTD".Dispositivo[#Maquina].Mov_Manual.Confirmar_Orden )
      S_Coil( "DB771_HMI_VTD".Dispositivo[#Maquina].Mov_Manual.Bussy )
   END_RUNG
   // the same network as SCL:
   #_w1 := #Estado_CBx.Manual_CBx AND "DB771_HMI_VTD".Dispositivo[#Maquina].Mov_Manual.Remoto_OK AND "DB771_HMI_VTD".Dispositivo[#Maquina].Mov_Manual.Enviar_Orden AND "DB771_HMI_VTD".Dispositivo[#Maquina].Mov_Manual.Confirmar_Orden AND NOT #Error_Tx;
   IF #_w1 THEN
       #Rem_MesaDestino := "DB771_HMI_VTD".Dispositivo[#Maquina].Mov_Manual.MesaDestino;
       #Rem_MesaOrigen := "DB771_HMI_VTD".Dispositivo[#Maquina].Mov_Manual.MesaHorquilla;
   END_IF;
   IF #_w1 AND (#Rem_MesaOrigen = "DB885_ConfigMaquinas".Maquina[#Maquina].Mesa_1) THEN
       #Posicion_Destino := "DB885_ConfigMaquinas".Maquina[#Maquina].Mesa[#Rem_MesaDestino].Posicion_mm_H1;
       #PeticionPiso_Activa := TRUE;
   END_IF;
   #_w2 := #_w1 AND (#Rem_MesaOrigen = "DB885_ConfigMaquinas".Maquina[#Maquina].Mesa_1);
   IF #_w2 THEN
       "DB771_HMI_VTD".Dispositivo[#Maquina].Mov_Manual.Enviar_Orden := FALSE;
       "DB771_HMI_VTD".Dispositivo[#Maquina].Mov_Manual.Confirmar_Orden := FALSE;
       "DB771_HMI_VTD".Dispositivo[#Maquina].Mov_Manual.Bussy := TRUE;
   END_IF;
   IF #_w1 AND (#Mesa_2 <> 0) AND (#Rem_MesaOrigen = "DB885_ConfigMaquinas".Maquina[#Maquina].Mesa_2) THEN
       #Posicion_Destino := "DB885_ConfigMaquinas".Maquina[#Maquina].Mesa[#Rem_MesaDestino].Posicion_mm_H2;
       #PeticionPiso_Activa := TRUE;
   END_IF;
   #_w3 := #_w1 AND (#Mesa_2 <> 0) AND (#Rem_MesaOrigen = "DB885_ConfigMaquinas".Maquina[#Maquina].Mesa_2);
   IF #_w3 THEN
       "DB771_HMI_VTD".Dispositivo[#Maquina].Mov_Manual.Enviar_Orden := FALSE;
       "DB771_HMI_VTD".Dispositivo[#Maquina].Mov_Manual.Confirmar_Orden := FALSE;
       "DB771_HMI_VTD".Dispositivo[#Maquina].Mov_Manual.Bussy := TRUE;
   END_IF;
END_REGION

REGION Network 22: Movimientos en Remoto - Reseteamos la orden cuando estamos en destino
   RUNG wire#powerrail
      Contact( #Estado_CBx.Manual_CBx )
      Contact( "DB771_HMI_VTD".Dispositivo[#Maquina].Mov_Manual.Remoto_OK )
      Contact( "DB951_InterlockMaquinas".Maquina[#Maquina].PosOK )
      wire#w1
      R_Coil( #PeticionPiso_Activa )
      R_Coil( "DB771_HMI_VTD".Dispositivo[#Maquina].Mov_Manual.Remoto_OK )
      R_Coil( "DB771_HMI_VTD".Dispositivo[#Maquina].Mov_Manual.Bussy )
   END_RUNG
   RUNG wire#w1
      Move(in := 0, out1 => "DB771_HMI_VTD".Dispositivo[#Maquina].Mov_Manual.MesaDestino, out2 => "DB771_HMI_VTD".Dispositivo[#Maquina].Mov_Manual.MesaHorquilla)
   END_RUNG
   // the same network as SCL:
   IF #Estado_CBx.Manual_CBx AND "DB771_HMI_VTD".Dispositivo[#Maquina].Mov_Manual.Remoto_OK AND "DB951_InterlockMaquinas".Maquina[#Maquina].PosOK THEN
       #PeticionPiso_Activa := FALSE;
   END_IF;
   #_w1 := #Estado_CBx.Manual_CBx AND "DB771_HMI_VTD".Dispositivo[#Maquina].Mov_Manual.Remoto_OK AND "DB951_InterlockMaquinas".Maquina[#Maquina].PosOK;
   IF #_w1 THEN
       "DB771_HMI_VTD".Dispositivo[#Maquina].Mov_Manual.Remoto_OK := FALSE;
       "DB771_HMI_VTD".Dispositivo[#Maquina].Mov_Manual.Bussy := FALSE;
       "DB771_HMI_VTD".Dispositivo[#Maquina].Mov_Manual.MesaDestino := 0;
       "DB771_HMI_VTD".Dispositivo[#Maquina].Mov_Manual.MesaHorquilla := 0;
   END_IF;
END_REGION

REGION Network 23: >>>>>>>>>>>>>>>>>>>>>>>>>>>>>>>>>>>>>>>>>>>>>>>>>>>>>>>>>>>>>>>>>>>>>>>>>>>>>>>>
END_REGION

REGION Network 24: SALIDAS
   RUNG wire#powerrail
      Contact( #Estado_CBx.Marcha_CBx )
      I_Contact( "DB951_InterlockMaquinas".Maquina[#Maquina].PosOK )
      I_Contact( #Error_Tx )
      { S7_Templates := "SrcType := Real" } GT_Contact(in1 := #Posicion_Destino, in2 := "DB885_ConfigMaquinas".Maquina[#Maquina].PosMinima)
      { S7_Templates := "SrcType := Real" } LT_Contact(in1 := #Posicion_Destino, in2 := "DB885_ConfigMaquinas".Maquina[#Maquina].PosMaxima)
      wire#w1
      Move(in := #Posicion_Destino, out1 => #PosicionDestino)
   END_RUNG
   RUNG wire#w1
      Contact( #PeticionPiso_Activa )
      Coil( #Orden )
   END_RUNG
   // the same network as SCL:
   #_w1 := #Estado_CBx.Marcha_CBx AND NOT "DB951_InterlockMaquinas".Maquina[#Maquina].PosOK AND NOT #Error_Tx AND (#Posicion_Destino > "DB885_ConfigMaquinas".Maquina[#Maquina].PosMinima) AND (#Posicion_Destino < "DB885_ConfigMaquinas".Maquina[#Maquina].PosMaxima);
   IF #_w1 THEN #PosicionDestino := #Posicion_Destino; END_IF;
   #Orden := #_w1 AND #PeticionPiso_Activa;
END_REGION
END_FUNCTION_BLOCK
